# EPICS autosave request: softGlueApp/Db/threshTrig_settings.req
$(P)$(H)threshTrig-$(N)_desc
$(P)$(H)threshTrig-$(N)_EN_Signal
$(P)$(H)threshTrig-$(N)_CLK_Signal
$(P)$(H)threshTrig-$(N)_TRIG_Signal
$(P)$(H)threshTrig-$(N)_POSTHR
$(P)$(H)threshTrig-$(N)_NEGTHR
